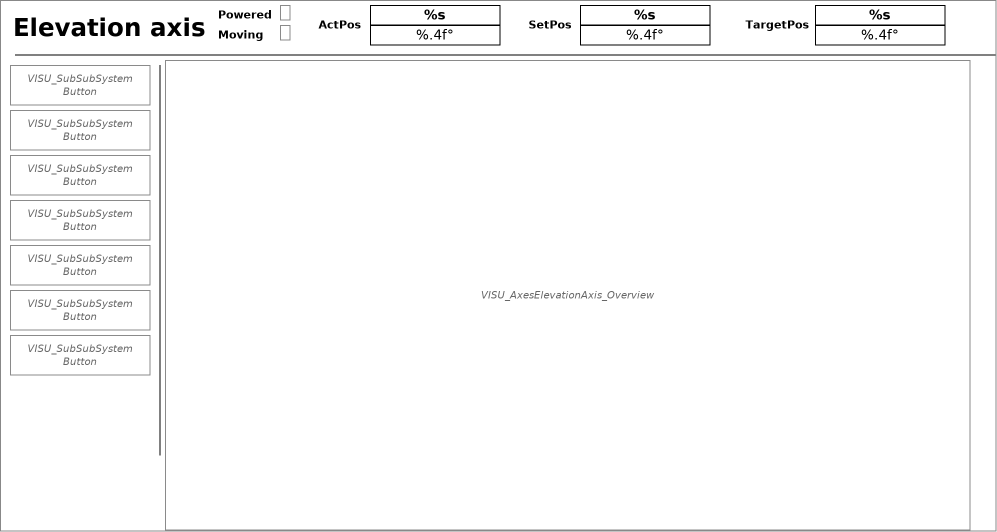
VISUALIZATION VISU_AxesElevationAxis  // 997x532
VAR_IN_OUT
	ref : AxesElevationAxis;
    ref_driveChannel : AX52XXDriveChannel;
    widget : AxesElevationAxisWidget;
END_VAR
    Rectangle (10,5 590x45), "Elevation axis"
    Frame (10,65 140x40)
        shows VISU_SubSubSystemButton(widget := widget.button_overview)
        OnMouseClick: FrameSelectionChange Selection=SelectedFrame=e720f99c-78fc-49d3-920d-5c22fdf0231f, GlobSel=AssignType=Directly, SelType=Locally
        OnMouseClick: execute { widget.activeTab := AxesElevationAxisTabs.OVERVIEW; }
    Frame (165,60 805x470)
        shows VISU_AxesElevationAxis_Overview(ref := ref, widget := widget)
        shows VISU_AxesElevationAxis_Processes(ref := ref, ref_driveChannel := ref_driveChannel, widget := widget)
        shows VISU_AX522DriveChannel(ref := ref_driveChannel, widget := widget.driveChannel)
        shows VISU_AngularAxis(axis := ref.parts.virtualAxis, widget := widget.virtualAxis)
        shows VISU_AngularAxis(axis := ref.parts.physicalAxis, widget := widget.physicalAxis)
        shows VISU_AxesElevationAxis_Lidas(ref := ref, widget := widget)
        shows VISU_AxesElevationAxis_AbsoluteEncoder(ref := ref, widget := widget)
        shows VISU_AxesAzimuthAxis_AbsoluteEncoder(ref := ref, widget := widget)
        p3523098516: ref
    Line (160,455) (160,65)
    Frame (10,155 140x40)
        shows VISU_SubSubSystemButton(widget := widget.button_driveChannel)
        OnMouseClick: FrameSelectionChange Selection=SelectedFrame=e720f99c-78fc-49d3-920d-5c22fdf0231f, Selection=2, GlobSel=AssignType=Directly, SelType=Locally
        OnMouseClick: execute { widget.activeTab := AxesElevationAxisTabs.DRIVE_CHANNEL; }
    Frame (10,200 140x40)
        shows VISU_SubSubSystemButton(widget := widget.button_virtualAxis)
        OnMouseClick: FrameSelectionChange Selection=SelectedFrame=e720f99c-78fc-49d3-920d-5c22fdf0231f, Selection=3, GlobSel=AssignType=Directly, SelType=Locally
        OnMouseClick: execute { widget.activeTab := AxesElevationAxisTabs.VIRTUAL_AXIS; }
    Frame (10,245 140x40)
        shows VISU_SubSubSystemButton(widget := widget.button_physicalAxis)
        OnMouseClick: FrameSelectionChange Selection=SelectedFrame=e720f99c-78fc-49d3-920d-5c22fdf0231f, Selection=4, GlobSel=AssignType=Directly, SelType=Locally
        OnMouseClick: execute { widget.activeTab := AxesElevationAxisTabs.PHYSICAL_AXIS; }
    Frame (10,290 140x40)
        shows VISU_SubSubSystemButton(widget := widget.button_lidas)
        OnMouseClick: FrameSelectionChange Selection=SelectedFrame=e720f99c-78fc-49d3-920d-5c22fdf0231f, Selection=5, GlobSel=AssignType=Directly, SelType=Locally
        OnMouseClick: execute { widget.activeTab := AxesElevationAxisTabs.LIDAS; }
    Frame (10,335 140x40)
        shows VISU_SubSubSystemButton(widget := widget.button_absoluteEncoder)
        OnMouseClick: FrameSelectionChange Selection=SelectedFrame=e720f99c-78fc-49d3-920d-5c22fdf0231f, Selection=6, GlobSel=AssignType=Directly, SelType=Locally
        OnMouseClick: execute { widget.activeTab := AxesElevationAxisTabs.ABSOLUTE_ENCODER; }
    Frame (10,110 140x40)
        shows VISU_SubSubSystemButton(widget := widget.button_processes)
        OnMouseClick: FrameSelectionChange Selection=SelectedFrame=e720f99c-78fc-49d3-920d-5c22fdf0231f, Selection=1, GlobSel=AssignType=Directly, SelType=Locally
        OnMouseClick: execute { widget.activeTab := AxesElevationAxisTabs.PROCESSES; }
    Line (995,55) (15,55)
    Label (310,0 60x50), "ActPos"
    Rectangle (370,5 130x20), "%s", text variable: widget.actPos.dmsString
    Rectangle (370,25 130x20), "%.4f°", text variable: ref.actPos.degrees.value
    Label (520,0 60x50), "SetPos"
    Rectangle (580,5 130x20), "%s", text variable: widget.setPos.dmsString
    Rectangle (580,25 130x20), "%.4f°", text variable: ref.setPos.degrees.value
    Label (740,0 75x50), "TargetPos"
    Rectangle (815,5 130x20), "%s", text variable: widget.targetPos.dmsString
    Rectangle (815,25 130x20), "%.4f°", text variable: ref.targetPos.degrees.value
    Label (215,5 65x20), "Powered"
    Frame (280,5 10x15)
        shows VISU_State_gray_green(state := ref.statuses.poweredStatus.enabled)
    Label (215,25 65x20), "Moving"
    Frame (280,25 10x15)
        shows VISU_State_gray_green(state := ref.parts.physicalAxis.axis_ref.Status.Moving)
END_VISUALIZATION

(* stored: Version 1.1.0.1, ProductVersion 3.1.4019.2
   Visu VISU_AxesElevationAxis: Id {f0334d99-a977-4bc5-a20b-a05d2cbde238} *)
